TYPE ST_SpeedProfile :
STRUCT
	fVelocity : LREAL := 10.0; 
	fAcceleration : LREAL := 100.0; 
	fDeceleration : LREAL := 100.0; 
	fJerk : LREAL := 1000.0;
END_STRUCT
END_TYPE

(* stored: Version 1.1.0.1, ProductVersion 3.1.4024.12
   DUT ST_SpeedProfile: Id {1d09f39f-6282-48e1-aaa5-ab1459d21499} *)
